FUNCTION_BLOCK TimeConvertor
VAR_INPUT
END_VAR
VAR_OUTPUT
END_VAR
VAR
END_VAR

METHOD fromfiletime64 : ST_TimeConvertor
VAR_INPUT
END_VAR
END_METHOD

END_FUNCTION_BLOCK

(* stored: Version 1.1.0.1, ProductVersion 3.1.4024.12
   POU TimeConvertor: Id {6f83ad14-afca-4c00-a094-9e62c095e8f5}, SpecialFunc None
   Method fromfiletime64: Id {f163be2f-78be-48cb-83b8-efa80460427c} *)
